GLOBALCONSTANTS DefaultPool_Numeric (* Numeric object pool constants (ID, Scale, Offset, Decimals) *)
  PACKAGE Uebungen::const::UT::HystereseHorizontal;
END_GLOBALCONSTANTS
